// LS Electric XG5000 project: HelloWorld
// PLC LSPLC

PROGRAM SimulatorTest (task: 스캔 프로그램)

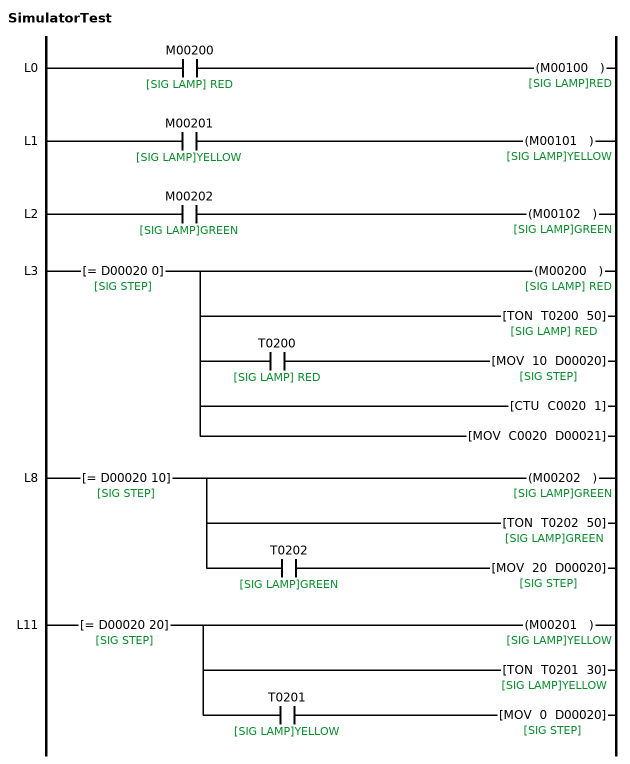
; L0
LOAD      M00200	// [SIG LAMP] RED
OUT       M00100	// [SIG LAMP]RED
; L1
LOAD      M00201	// [SIG LAMP]YELLOW
OUT       M00101	// [SIG LAMP]YELLOW
; L2
LOAD      M00202	// [SIG LAMP]GREEN
OUT       M00102	// [SIG LAMP]GREEN
; L3
LOAD=     D00020 0	// [SIG STEP]
OUT       M00200	// [SIG LAMP] RED
TON       T0200 50	// [SIG LAMP] RED
MPUSH
AND       T0200	// [SIG LAMP] RED
MOV       10 D00020	// [SIG STEP]
MPOP
CTU       C0020 1
MOV       C0020 D00021
; L8
LOAD=     D00020 10	// [SIG STEP]
OUT       M00202	// [SIG LAMP]GREEN
TON       T0202 50	// [SIG LAMP]GREEN
AND       T0202	// [SIG LAMP]GREEN
MOV       20 D00020	// [SIG STEP]
; L11
LOAD=     D00020 20	// [SIG STEP]
OUT       M00201	// [SIG LAMP]YELLOW
TON       T0201 30	// [SIG LAMP]YELLOW
AND       T0201	// [SIG LAMP]YELLOW
MOV       0 D00020	// [SIG STEP]

VARIABLES AND COMMENTS (devices not used above)
M0100	WORD	[SIG STEP]